// TIA Portal V17 export
// export: Created 2023-02-13T11:16:43.5023678Z, ExportSetting WithDefaults, DisplayName Totally Integrated Automation Portal, DisplayVersion V17, DisplayName TIA Portal Openness, DisplayVersion V17, DisplayName TIA Portal Teamcenter Gateway, DisplayVersion V17, DisplayName TIA Portal Version Control Interface, DisplayVersion V17, DisplayName SINAMICS Startdrive Advanced, DisplayVersion V17, DisplayName SINAMICS Startdrive G130, G150, S120, S150, SINAMICS MV, S210, DisplayVersion V17, DisplayName SINAMICS Startdrive G110M, G120, G120C, G120D, G120P, G115D, DisplayVersion V17, DisplayName STEP 7 Professional, DisplayVersion V17, DisplayName STEP 7 Safety, DisplayVersion V17, DisplayName WinCC Professional, DisplayVersion V17
DATA_BLOCK "T-85.00"   // DB52
VERSION : 0.1
// stored: AutoNumber false, DBAccessibleFromOPCUA true, DBAccessibleFromWebserver true, InstanceOfName Storage_Tank_Multi_Inload, InstanceOfType FB
"Storage_Tank_Multi_Inload"
   // VAR_INPUT
   //    Level_Bypass : Bool;
   //    Single_CIP_Cmd : Bool;
   //    IN_FBAV_Load : Bool;
   //    IN_FBAV_Transfer : Bool;
   //    IN_FBP_Transfer : Bool;
   //    IN_FBP_Transfer_Speed : Real;
   //    IN_FBP_CIP : Bool;
   //    IN_FBAV_CIP_Sup : Bool;
   //    IN_FBAV_CIP_Tank : Bool;
   //    IN_FBAV_CIP_Line : Bool;
   //    IN_LT01 : Real;
   //    IN_FS : Bool;
   //    CIP_Req_OK : Bool;
   //    CIP_ON_Progress : Bool;
   //    CIP_Supply_ON : Bool;
   //    CIP_Complete : Bool;
   //    CIPPulse : Bool;
   //    Filler_Product_Req : Bool;
   //    Filler_CIP_Req : Bool;
   //    Loading_Busy_1 : Bool;
   //    Loading_Busy_2 : Bool;
   //    Loading_Busy_3 : Bool;
   //    Transfer_Busy : Bool;
   //    CIP_En : Bool;
   // END_VAR
   // VAR_OUTPUT
   //    Out_AV_Load : Bool;
   //    Out_AV_Transfer : Bool;
   //    Out_P_Transfer : Bool;
   //    Out_P_TF_Speed : Real;
   //    Out_P_CIP : Bool;
   //    Out_AV_CIP_Line : Bool;
   //    Out_AV_CIP_Tank : Bool;
   //    Out_AV_CIP_Filling : Bool;
   //    CIP_Tank_Req : Bool;
   //    CIP_Line_Req : Bool;
   //    CIP_LineOK : Bool;
   // END_VAR
   // VAR
   //    Cmd : Struct
   //       Inload_Select_Tank_1 : Bool;
   //       Inload_Select_Tank_2 : Bool;
   //       Inload_Select_Tank_3 : Bool;
   //       Inload : Bool;
   //       Tank_CIP_Req : Bool;
   //       Line_CIP_Req : Bool;
   //       Tank_Filling_CIP_Req : Bool;
   //       CIP_Filling_En : Bool;
   //       CIP_Line_Req_OK : Bool;
   //       CIP_Supply_ON : Bool;
   //       CIP_ON_Progress : Bool;
   //       Flushing : Bool;
   //       RaadyForTF : Bool;
   //       Flush_Select : Byte;
   //       Drain_In : Bool;
   //       Drain_Transfer : Bool;
   //    END_STRUCT;
   //    Param : Struct
   //       SP_Level_LL : Real;
   //       SP_Level_ML : Real;
   //       SP_Level_HL : Real;
   //       SupplyPump_SP_Speed : Real;
   //       L_Hi_Lim : Real;
   //       L_Lo_Lim : Real;
   //       L_Hys : Real;
   //       FlushingTime : DInt;
   //       CIP_Trf_SP_Speed : Real;
   //       CIP_Ret_ON_SP : Real;
   //       CIP_Ret_OFF_SP : Real;
   //       Transfer_P_Speed : Real;
   //       Drain_Inload_SP : DInt;
   //       Drain_Transfer_SP : DInt;
   //       SP_Agi_On : Real;
   //    END_STRUCT;
   //    State : Struct
   //       Tank_inloading : Bool;
   //       Tank_inCIP : Bool;
   //       Tank_Filling_inCIP : Bool;
   //       Line_inCIP : Bool;
   //       FIlling_inCIP : Bool;
   //       Flushing : Bool;
   //       Tank_LL : Bool;
   //       Tank_ML : Bool;
   //       Tank_HL : Bool;
   //       Inload_Enable : Bool;
   //       Tank_CIP_Enable : Bool;
   //       Line_CIP_Enable : Bool;
   //       Tank_Filling_CIP_Enable : Bool;
   //       Flushing_Enable : Bool;
   //       Flush_selected : Byte;
   //       CIP_Request_OK : Bool;
   //       CIP_ReturnON : Bool;
   //       Ready_For_Transfer_EN : Bool;
   //       Ready_For_Transfer : Bool;
   //       HWT_Status : Int;
   //       Transfer_to_Filling : Bool;
   //       "Line_AV4&AV5" : Bool;
   //       "Line_AV1&AV2" : Bool;
   //       "Line_AV7&AV8" : Bool;
   //       "Line_AV10&AV11" : Bool;
   //       "Line_AV5&AV6" : Bool;
   //       CIP_Line1_ON : Bool;
   //       CIP_Line2_ON : Bool;
   //       CIP_Line3_ON : Bool;
   //       CIP_Line4_ON : Bool;
   //       Drain_Inload : Bool;
   //       Drain_Transfer : Bool;
   //       Agi_ON : Bool;
   //       "CIP Req" : Bool;
   //    END_STRUCT;
   //    alwaysON : Bool;
   //    L_Hys_Abs : Real;
   //    Hys_Level_HL : Real;
   //    Hys_Level_ML : Real;
   //    Hys_Level_LL : Real;
   //    Drain_Inload_MSec : DInt;
   //    Drain_Inload_Count : IEC_DCOUNTER;
   //    Drain_Inload_Act { S7_SetPoint := 'True'} : DInt;
   //    Drain_Transfer_MSec : DInt;
   //    Drain_Transfer_Count : IEC_DCOUNTER;
   //    Drain_Transfer_Act : DInt;
   //    r : Struct
   //       PosE1 : Bool;
   //       PosE2 : Bool;
   //       PosE3 : Bool;
   //       PosE4 : Bool;
   //       PosE5 : Bool;
   //       PosE6 : Bool;
   //       PosE7 : Bool;
   //       PosE8 : Bool;
   //       PosE9 : Bool;
   //       PosE10 : Bool;
   //       PosE11 : Bool;
   //       PosE12 : Bool;
   //       PosE13 : Bool;
   //       PosE14 : Bool;
   //       PosE15 : Bool;
   //       PosE16 : Bool;
   //       PosE17 : Bool;
   //       PosE18 : Bool;
   //       PosE19 : Bool;
   //       PosE20 : Bool;
   //       PosE21 : Bool;
   //       PosE22 : Bool;
   //       PosE23 : Bool;
   //       PosE24 : Bool;
   //       PosE25 : Bool;
   //       PosE26 : Bool;
   //       PosE27 : Bool;
   //       PosE28 : Bool;
   //       PosE29 : Bool;
   //       PosE30 : Bool;
   //       PosE31 : Bool;
   //       PosE32 : Bool;
   //    END_STRUCT;
   //    Actuator : Struct
   //       AV_Outlet : Bool;
   //       AV_Load : Bool;
   //       AV_Transfer : Bool;
   //       CIP_Line_Pump : Bool;
   //       CIP_Tank_Pump : Bool;
   //       TransferPump : Bool;
   //       FlushPump : Bool;
   //       CV_Steam : Bool;
   //       Pump : Bool;
   //    END_STRUCT;
   //    SPumpTim { S7_SetPoint := 'True'} : TON_TIME;
   //    SAV_CIPLine { S7_SetPoint := 'True'} : TON_TIME;
   //    SAV_CIPTANK { S7_SetPoint := 'True'} : TON_TIME;
   //    SAV_CIPFILLING { S7_SetPoint := 'True'} : TON_TIME;
   //    AVinloadTim { S7_SetPoint := 'True'} : TON_TIME;
   //    AVOutletTim { S7_SetPoint := 'True'} : TON_TIME;
   //    Drain_In_Tim { S7_SetPoint := 'True'} : TON_TIME;
   //    Drain_Out_Tim { S7_SetPoint := 'True'} : TON_TIME;
   //    "Pump Off Tim" { S7_SetPoint := 'True'} : TON_TIME;
   //    "Loading_Busy Tim_1" { S7_SetPoint := 'True'} : TON_TIME;
   //    "Loading_Busy Tim_2" { S7_SetPoint := 'True'} : TON_TIME;
   //    "Loading_Busy Tim_3" { S7_SetPoint := 'True'} : TON_TIME;
   //    Hys_Level_Agi { S7_SetPoint := 'True'} : Real;
   // END_VAR
BEGIN
END_DATA_BLOCK
